(*
SPDX-FileCopyrightText: © 2026 Oleksandr Tiutyk <trofimich@gmail.com>
SPDX-License-Identifier: MIT
License: https://opensource.org/license/mit
*)

(*!
<summary>Base automation component representing a leaf node in the component hierarchy.</summary>
<description>
Leaf components have no children and represent terminal devices, sensors, or actuators.
Events received at this level bubble upwards to the parent component unless propagation is stopped.
Lifecycle methods execute leaf-specific state transitions and invoke overridable hooks. Parent is mandatory
and borrowed for the leaf lifetime. It is checked before initialization hooks. Use one owner task per instance.
Execute() can recover the stored non-critical execution error. Descendants can defer recovery until its
cause clears and can report other diagnostics independently.
</description>
*)

FUNCTION_BLOCK ABSTRACT LeafAutomationComponent EXTENDS AutomationComponent IMPLEMENTS IChildAutomationComponent
VAR
	{attribute 'hide'} 
	_Parent : IParentAutomationComponent;
END_VAR

(*!
<summary>Dispatches event locally and bubbles it up to the parent component.</summary>
<param name="event">The event to dispatch.</param>
*)
METHOD FINAL BubbleEvent
VAR_INPUT
	event : TOF_Core.IEvent;
END_VAR
VAR
	stopPropagation : BOOL;
	
	parentAsBubbleEventDispatcher : TOF_Core.IBubbleEventDispatcher;
END_VAR
OnEventReceived(event := event, stopPropagation => stopPropagation);

IF stopPropagation THEN
	RETURN;
END_IF

IF __QUERYINTERFACE(Parent, parentAsBubbleEventDispatcher) THEN
	parentAsBubbleEventDispatcher.BubbleEvent(event := event);
END_IF
END_METHOD

(*!
<summary>Reports whether Execute() can clear a pending non-critical execution error.</summary>
<description>
The base allows immediate recovery. A descendant can defer recovery by returning FALSE. Execute() calls
this only in WORKING with an active non-critical execution error. Returning FALSE retains the diagnostic
and allows OnWorking to run. Overrides must observe current state without side effects or exceptions.
</description>
*)
METHOD PROTECTED CanRecoverExecutionError : BOOL
CanRecoverExecutionError := TRUE;
END_METHOD

(*!
<summary>Disables the leaf component and invokes OnDisable.</summary>
*)
METHOD FINAL Disable
VAR
	exceptionCode : __SYSTEM.ExceptionCode;
END_VAR
VAR_INST
	disabling : BOOL;
END_VAR
IF NOT _Enabled OR_ELSE disabling THEN
	RETURN;
END_IF

disabling := TRUE;

__TRY
	OnDisable();
	
	_Enabled := FALSE;
	
	disabling := FALSE;	
__CATCH(exceptionCode)
	disabling := FALSE;
	
	TOF_Core.ExceptionManager.ReThrowLastException(
		exceptionCode := exceptionCode,
		catchPointNamespaceName := NamespaceName,
		catchPointPOUName := __POUNAME(),
		catchPointPosition := __POSITION()
	);
__ENDTRY
END_METHOD

(*!
<summary>Enables the leaf component and invokes OnEnable.</summary>
<description>
Enabling does not automatically reset a STOPPED leaf; a disabled stopped leaf remains STOPPED after Enable
until explicitly Reset. If the parent is disabled, enables the parent with includeChildren := FALSE.
</description>
<param name="includeChildren">Ignored for leaf components as they have no children.</param>
*)
METHOD FINAL Enable
VAR_INPUT
	includeChildren : BOOL := TRUE;
END_VAR
VAR
	exceptionCode : __SYSTEM.ExceptionCode;
END_VAR
VAR_INST
	enabling : BOOL;
END_VAR
IF _Enabled OR_ELSE enabling THEN
	RETURN;
END_IF

enabling := TRUE;

__TRY
	OnEnable();
	
	IF _Parent <> 0 AND_THEN NOT _Parent.Enabled THEN
		_Parent.Enable(includeChildren := FALSE);
	END_IF
	
	_Enabled := TRUE;
	
	enabling := FALSE;
__CATCH(exceptionCode)
	enabling := FALSE;
	
	TOF_Core.ExceptionManager.ReThrowLastException(
		exceptionCode := exceptionCode,
		catchPointNamespaceName := NamespaceName,
		catchPointPOUName := __POUNAME(),
		catchPointPosition := __POSITION()
	);
__ENDTRY
END_METHOD

(*!
<summary>Advances cyclic execution for an enabled WORKING or STOPPED leaf.</summary>
<description>
In WORKING, checks CanRecoverExecutionError() for a pending non-critical execution error. When ready,
clears that record and invokes OnRecover before OnWorking. An exception during recovery always records
a copied CRITICAL error, stops the leaf without consulting ExceptionHandlingPolicy, and skips OnWorking.
In STOPPED, invokes OnStopped on each Execute call and logs failures.
</description>
*)
{attribute 'estimated-stack-usage' := '99'}
METHOD FINAL Execute
VAR
	exceptionCode : __SYSTEM.ExceptionCode;
	exception : TOF_Core.IException;	
	exceptionReaction : TOF_Core.EXCEPTION_REACTION;
END_VAR

IF NOT Enabled
	OR_ELSE (_OperationalState <> OPERATIONAL_STATE.WORKING AND_THEN _OperationalState <> OPERATIONAL_STATE.STOPPED)
THEN
	RETURN;
END_IF

CASE _OperationalState OF
	OPERATIONAL_STATE.WORKING:
		IF _Error.HasError AND_THEN _Error.Severity <> TOF_Core.ERROR_SEVERITY.CRITICAL THEN
			__TRY
				IF CanRecoverExecutionError() THEN
					_Error.Clear();
					OnRecover();
				END_IF
			__CATCH(exceptionCode)		
				exception := TOF_Core.ExceptionManager.GetLastException(
					exceptionCode := exceptionCode,
					catchPointNamespaceName := NamespaceName,
					catchPointPOUName := __POUNAME(),
					catchPointPosition := __POSITION()
				);

				// A recovery failure stops the leaf with a critical error without consulting the policy.
				ProcessException(
					exception := exception,
					exceptionReaction := TOF_Core.EXCEPTION_REACTION.SET_ERROR_AND_STOP,
					exceptionSourceHint := "OnRecover error"
				);

				RETURN;
			__ENDTRY
		END_IF
		
		__TRY
			OnWorking();
		__CATCH(exceptionCode)
			exception := TOF_Core.ExceptionManager.GetLastException(
				exceptionCode := exceptionCode,
				catchPointNamespaceName := NamespaceName,
				catchPointPOUName := __POUNAME(),
				catchPointPosition := __POSITION()
			);	
		
			exceptionReaction := OnHandleException(exception := exception, failedMethodName := 'OnWorking');
		
			ProcessException(
				exception := exception,
				exceptionReaction := exceptionReaction,
				exceptionSourceHint := "OnWorking error"
			);
		
			IF exceptionReaction = TOF_Core.EXCEPTION_REACTION.SET_ERROR_AND_STOP THEN
				RETURN;		
			END_IF
		__ENDTRY
		
	OPERATIONAL_STATE.STOPPED:
		__TRY
			OnStopped();
		__CATCH(exceptionCode)
			exception := TOF_Core.ExceptionManager.GetLastException(
				exceptionCode := exceptionCode,
				catchPointNamespaceName := NamespaceName,
				catchPointPOUName := __POUNAME(),
				catchPointPosition := __POSITION()
			);	
		
			exceptionReaction := OnHandleException(exception := exception, failedMethodName := 'OnStopped');
		
			TOF_Core.LogManager.TryLogException(
				exception := exception,
				severity := GetErrorSeverityByExceptionReaction(exceptionReaction := exceptionReaction),
				topic1 := "AutomationComponent",
				topic2 := "AutomationComponent.OnStopped"
			);
		__ENDTRY	
END_CASE
END_METHOD

(*!
<summary>Initializes a new instance of the leaf component.</summary>
<param name="name">Descriptive name of the component.</param>
<param name="parent">Parent automation component in the hierarchy.</param>
*)
METHOD FB_init : BOOL
VAR_INPUT
	bInitRetains : BOOL; // TRUE: the retain variables are initialized (reset warm / reset cold)
	bInCopyCode : BOOL;  // TRUE: the instance will be copied to the copy code afterward (online change)
	name : WSTRING;
	parent : IParentAutomationComponent;
END_VAR
_Parent := parent;
END_METHOD

(*!
<summary>Validates the parent and advances leaf-specific initialization.</summary>
<description>
Parent is mandatory and borrowed for the leaf lifetime. Missing Parent fails before OnInitializing,
even if that hook would complete immediately. FALSE reports pending work or a caught failure; failures
record a critical error in terminal INVALID. TRUE reports completed initialization, including an already
stopped leaf. Completed hook effects are not rolled back.
</description>
*)
METHOD FINAL Initialize : BOOL
VAR
	exceptionCode : __SYSTEM.ExceptionCode;
	exception : TOF_Core.IException;
	
END_VAR
IF _OperationalState <> OPERATIONAL_STATE.INITIALIZING THEN
	Initialize := _OperationalState <> OPERATIONAL_STATE.INVALID;
	
	RETURN;
END_IF

__TRY
	IF _Parent = 0 THEN
		TOF_Core.Exceptions.ThrowDataMemberNotSpecified(
			sourceNamespaceName := NamespaceName,
			sourceClassName := ClassName,
			sourcePOUName := __POUNAME(),
			sourcePosition := __POSITION(),
			dataMemberName := 'Parent'
		);
	END_IF

	Initialize := OnInitializing();
	
	IF Initialize THEN
		SetOperationalState(state := OPERATIONAL_STATE.WORKING, reason := "Successfull initialization");
	ELSE
		IF _InitializationTimer.PT = T#0S THEN
			_InitializationTimer.PT := Parameters.InitializationTimeout;
		END_IF
		
		_InitializationTimer(IN := TRUE);
		
		IF _InitializationTimer.Q THEN		
			TOF_Core.Exceptions.ThrowTimeout(
				sourceNamespaceName := NamespaceName,
				sourceClassName := ClassName,
				sourcePOUName := __POUNAME(),
				sourcePosition := __POSITION(),
				timeoutValue := _InitializationTimer.PT,
				operationName := "Initialization"
			);
		END_IF
		
	END_IF	
__CATCH(exceptionCode)
	Initialize := FALSE;

	exception := TOF_Core.ExceptionManager.GetLastException(
		exceptionCode := exceptionCode,
		catchPointNamespaceName := NamespaceName,
		catchPointPOUName := __POUNAME(),
		catchPointPosition := __POSITION()
	);
	
	ProcessException(
		exception := exception,
		exceptionReaction := TOF_Core.EXCEPTION_REACTION.SET_ERROR_AND_CONTINUE,
		exceptionSourceHint := "Initialization error"
	);					
__ENDTRY
END_METHOD

(*!
<summary>Hook invoked when the leaf component is disabled.</summary>
*)
METHOD PROTECTED OnDisable
END_METHOD

(*!
<summary>Hook invoked when the leaf component is enabled.</summary>
*)
METHOD PROTECTED OnEnable
END_METHOD

(*!
<summary>Hook invoked to perform custom initialization for the leaf component.</summary>
<description>Returns TRUE when initialization completes successfully.</description>
*)
METHOD PROTECTED OnInitializing : BOOL
OnInitializing := TRUE;
END_METHOD

(*!
<summary>Hook invoked when the leaf component is reset from an error state.</summary>
*)
METHOD PROTECTED OnReset
END_METHOD

(*!
<summary>Hook invoked when the leaf component stops execution.</summary>
*)
METHOD PROTECTED OnStopped
END_METHOD

(*!
<summary>Hook invoked during cyclic execution when the leaf component is in the WORKING state.</summary>
*)
METHOD PROTECTED OnWorking
END_METHOD

(*!
<summary>Borrows the constructor-bound parent automation component.</summary>
<description>
Parent is mandatory for initialization and must remain live for the leaf lifetime. The getter does not
transfer ownership or permit reassignment.
</description>
*)
{attribute 'monitoring' := 'call'}
PROPERTY FINAL Parent : IParentAutomationComponent
GET
Parent := _Parent;
END_GET
END_PROPERTY

(*!
<summary>Resets the leaf component from an error state and transitions back to WORKING.</summary>
<description>
Served only while Enabled and STOPPED. Clears the execution error before invoking OnReset. If OnReset raises
an exception, the leaf remains STOPPED with a copied CRITICAL error without consulting ExceptionHandlingPolicy.
Completed hook effects are not rolled back.
</description>
*)
METHOD FINAL Reset
VAR
	exceptionCode : __SYSTEM.ExceptionCode;
	exception : TOF_Core.IException;	
END_VAR
IF NOT Enabled OR_ELSE _OperationalState <> OPERATIONAL_STATE.STOPPED THEN
	RETURN;
END_IF

_Error.Clear();

__TRY
	OnReset();
	
	SetOperationalState(state := OPERATIONAL_STATE.WORKING, reason := "Reset");
__CATCH(exceptionCode)		
	exception := TOF_Core.ExceptionManager.GetLastException(
		exceptionCode := exceptionCode,
		catchPointNamespaceName := NamespaceName,
		catchPointPOUName := __POUNAME(),
		catchPointPosition := __POSITION()
	);

	// A failed reset always keeps the leaf STOPPED with a critical error; the exception policy is not consulted.
	ProcessException(
		exception := exception,
		exceptionReaction := TOF_Core.EXCEPTION_REACTION.SET_ERROR_AND_STOP,
		exceptionSourceHint := "OnReset error"
	);
__ENDTRY
END_METHOD

(*!
<summary>Stops the leaf component and transitions to the STOPPED state.</summary>
<description>
Transitions a WORKING leaf to OPERATIONAL_STATE.STOPPED regardless of Enabled.
</description>
<param name="reason">Descriptive reason for stopping.</param>
*)
METHOD FINAL Stop
VAR_INPUT
	reason : WSTRING(255) := "External stop";
END_VAR
IF _OperationalState <> OPERATIONAL_STATE.WORKING THEN
	RETURN;
END_IF

SetOperationalState(state := OPERATIONAL_STATE.STOPPED, reason := reason);
END_METHOD

END_FUNCTION_BLOCK

(* stored: Version 1.1.0.1
   POU LeafAutomationComponent: Id {7c21300f-1ad4-4217-9d49-d0f060249ecb}, SpecialFunc None
   Folder Methods to override: Id {ca4cde0e-9a44-45fe-a0e4-7b7ca4e0c8a7}
   Method BubbleEvent: Id {42cce6a6-4219-41f5-a23e-d08f59aa4482}
   Method CanRecoverExecutionError: Id {48c1b0e0-7803-454f-9bc7-2cc9f5c9719b}
   Method Disable: Id {e7be34cc-e7d9-4568-8b6a-522ee606d568}
   Method Enable: Id {f7b45f9a-e580-4c1c-b27c-81b9ee1ab687}
   Method Execute: Id {54d74276-cad2-4fd8-8917-0010f6191e07}
   Method FB_init: Id {3ffe21cc-32bd-4767-9934-eaac8121d03b}
   Method Initialize: Id {3f657450-0a0b-4d21-8c85-c39655b515b8}
   Method OnDisable: Id {da5e244e-35a1-47cd-8144-7c7c3577035d}
   Method OnEnable: Id {7ab79cf0-ed24-4ab4-b074-f58d9b879980}
   Method OnInitializing: Id {87d0edb2-3f9d-4cdc-be5a-51ee4854c5ea}
   Method OnReset: Id {1437f653-2dca-4516-a643-9a7052ba8f91}
   Method OnStopped: Id {38cbad82-8eb7-4619-bb79-98729012ae5d}
   Method OnWorking: Id {02692fef-98a0-451c-b7a8-b233e155c1c5}
   Property Parent: Id {8fb3d4d7-c400-4c92-9c99-1346029f28e7}
   Get Get: Id {91af78c8-f2e0-4384-ac9d-b26f89ba6059}
   Method Reset: Id {39108ecc-e8fc-41d2-84a8-8d829dba9e49}
   Method Stop: Id {73828ae5-99ee-4c51-a656-702f6c6b2044} *)
